TYPE ST_CX_EL6080DataOut :
STRUCT
	nControl		: UINT;
	arrData			: ARRAY[0..1277] OF BYTE;
END_STRUCT
END_TYPE

(* stored: Version 1.1.0.1, ProductVersion 3.1.4024.15
   DUT ST_CX_EL6080DataOut: Id {41142290-0554-4710-b4fe-1f911e42e8dd} *)
